# EPICS autosave request: iocBoot/ioc13ide_linux/auto_settings.req
file "scaler_settings.req",             P=$(P), S=scaler1
file "SR570preamp_settings.req",        P=$(P), A=A1
file "SR570preamp_settings.req",        P=$(P), A=A2
file "SR570preamp_settings.req",        P=$(P), A=A3
file "SR570preamp_settings.req",        P=$(P), A=A4
file "scan_settings.req",               P=$(P), S=scan1
file "scan_settings.req",               P=$(P), S=scan2
file "scan_settings.req",               P=$(P), S=scan3
file "scan_settings.req",               P=$(P), S=scan4
file "saveData_settings.req"            P=$(P)
file "USB1808_settings.req", P=$(P1808)
file "USB3104_settings.req", P=$(P3104)
file "USBCTR_settings.req",  P=$(PCTR), MP=$(MP), SP=$(SP)
file "calc_GSECARS.req",                P=$(P)
file "Galil_settings.req",              P=$(P)
